(* Logix 5000 project; controller PLC2_Project_4_ServoApplication Emulate 5570 rev 20.11; software revision 20.00 *)
// A modular water treatment control system. Servo motor is connected to a cam/valve.

TASK MainTask (continuous, watchdog 500 ms) : MainProgram

MODULES
   Local : Emulate 5570 (ICP 1, rev 20.11)
      NicksIO : vendor 1 type 0 code 15 (ICP 2, rev 1.1, Output RPI 5 ms)
END_MODULES

PROGRAM MainProgram   (* main routine MainRoutine *)
VAR
   Button_CycleResetRequest : BOOL;
   Button_RequestCycle : BOOL;
   Cycle_Position : DINT := 4;   // Cycle Position/Mode 0 = Home 1 = Fill 2 = Drain 3 = Flush 4 = Travelling
   Cycle_Sequence : DINT := 3;   // Cycle Mode: SEQ 0 - FILL SEQ 1 - DRAIN SEQ 2 - FLUSH SEQ 3 - HOME
   DrainPosition_Delay : TIMER := (PRE := 20000);   // Drain position for 20 seconds
   FillPosition_Delay : TIMER := (PRE := 10000);   // Fill Position for 10 seconds
   FlushPosition_Delay : TIMER := (PRE := 10000);
   ONS_RequestCycle : BOOL;
   ONS_ResetRequest : BOOL;
   Servo_En : BOOL := 1;
   Switch_DrainPos : BOOL;
   Switch_FillPos : BOOL;
   Switch_FlushPos : BOOL;
   Switch_HomePos : BOOL;
END_VAR

ROUTINE Control   (* ladder *)
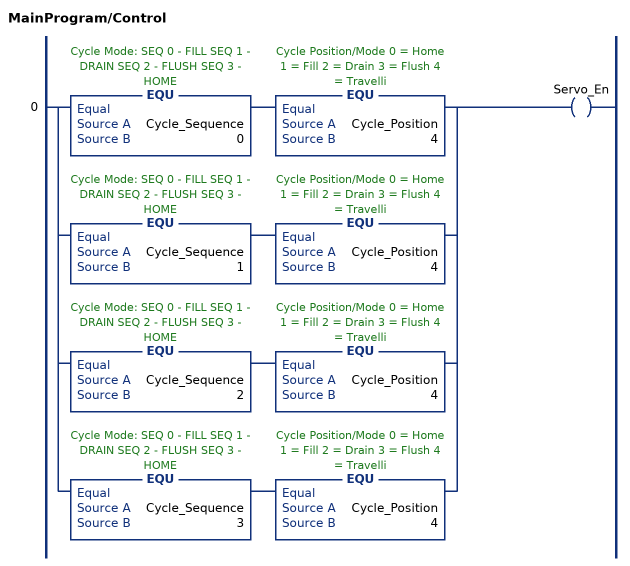
   0: [EQU(Cycle_Sequence,0) EQU(Cycle_Position,4) ,EQU(Cycle_Sequence,1) EQU(Cycle_Position,4) ,EQU(Cycle_Sequence,2) EQU(Cycle_Position,4) ,EQU(Cycle_Sequence,3) EQU(Cycle_Position,4) ]OTE(Servo_En);
END_ROUTINE

ROUTINE Cycle_Position   (* ladder *)
// What position is the valve in?
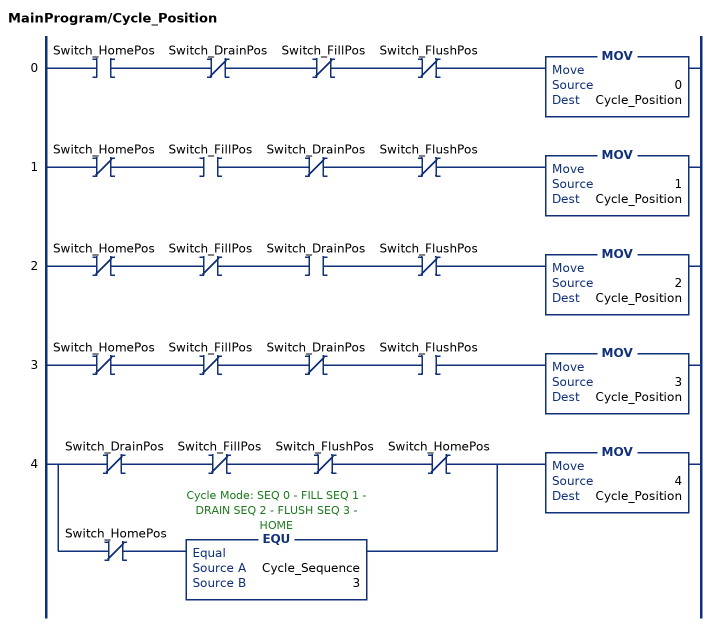
   0: XIC(Switch_HomePos)XIO(Switch_DrainPos)XIO(Switch_FillPos)XIO(Switch_FlushPos)MOV(0,Cycle_Position);
   1: XIO(Switch_HomePos)XIC(Switch_FillPos)XIO(Switch_DrainPos)XIO(Switch_FlushPos)MOV(1,Cycle_Position);
   2: XIO(Switch_HomePos)XIO(Switch_FillPos)XIC(Switch_DrainPos)XIO(Switch_FlushPos)MOV(2,Cycle_Position);
   3: XIO(Switch_HomePos)XIO(Switch_FillPos)XIO(Switch_DrainPos)XIC(Switch_FlushPos)MOV(3,Cycle_Position);
   4: [XIO(Switch_DrainPos) XIO(Switch_FillPos) XIO(Switch_FlushPos) XIO(Switch_HomePos) ,XIO(Switch_HomePos) EQU(Cycle_Sequence,3) ]MOV(4,Cycle_Position);
END_ROUTINE

ROUTINE Cycle_Sequence   (* ladder *)
// What stage in the cycle is the valve in?
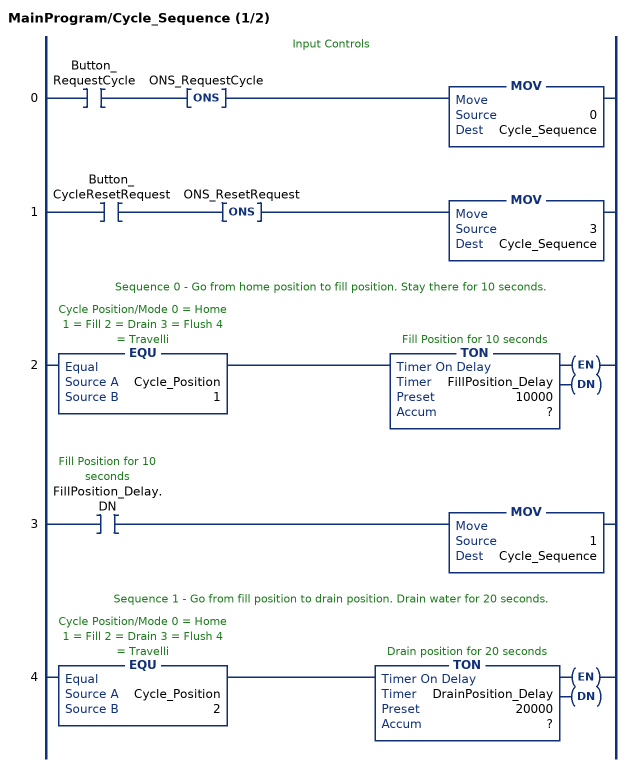
   // Input Controls
   0: XIC(Button_RequestCycle)ONS(ONS_RequestCycle)MOV(0,Cycle_Sequence);
   1: XIC(Button_CycleResetRequest)ONS(ONS_ResetRequest)MOV(3,Cycle_Sequence);
   // Sequence 0 - Go from home position to fill position. Stay there for 10 seconds.
   2: EQU(Cycle_Position,1)TON(FillPosition_Delay,?,?);
   3: XIC(FillPosition_Delay.DN)MOV(1,Cycle_Sequence);
   // Sequence 1 - Go from fill position to drain position. Drain water for 20 seconds.
   4: EQU(Cycle_Position,2)TON(DrainPosition_Delay,?,?);
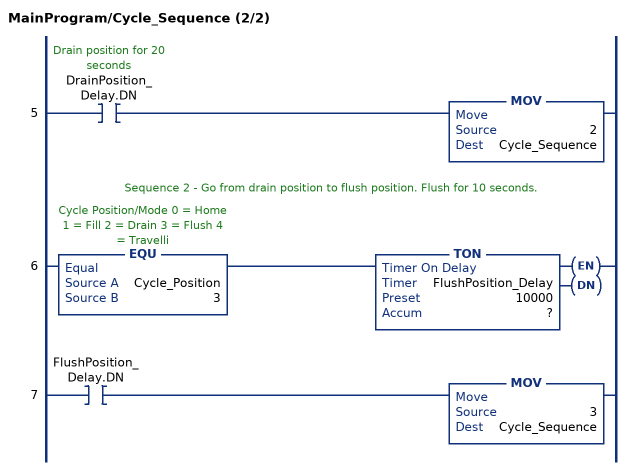
   5: XIC(DrainPosition_Delay.DN)MOV(2,Cycle_Sequence);
   // Sequence 2 - Go from drain position to flush position. Flush for 10 seconds.
   6: EQU(Cycle_Position,3)TON(FlushPosition_Delay,?,?);
   7: XIC(FlushPosition_Delay.DN)MOV(3,Cycle_Sequence);
END_ROUTINE

ROUTINE InputOutput   (* ladder *)
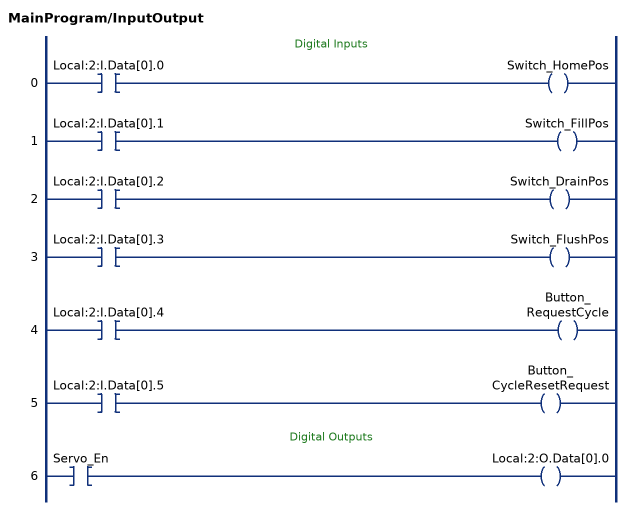
   // Digital Inputs
   0: XIC(Local:2:I.Data[0].0)OTE(Switch_HomePos);
   1: XIC(Local:2:I.Data[0].1)OTE(Switch_FillPos);
   2: XIC(Local:2:I.Data[0].2)OTE(Switch_DrainPos);
   3: XIC(Local:2:I.Data[0].3)OTE(Switch_FlushPos);
   4: XIC(Local:2:I.Data[0].4)OTE(Button_RequestCycle);
   5: XIC(Local:2:I.Data[0].5)OTE(Button_CycleResetRequest);
   // Digital Outputs
   6: XIC(Servo_En)OTE(Local:2:O.Data[0].0);
END_ROUTINE

ROUTINE MainRoutine   (* ladder *)
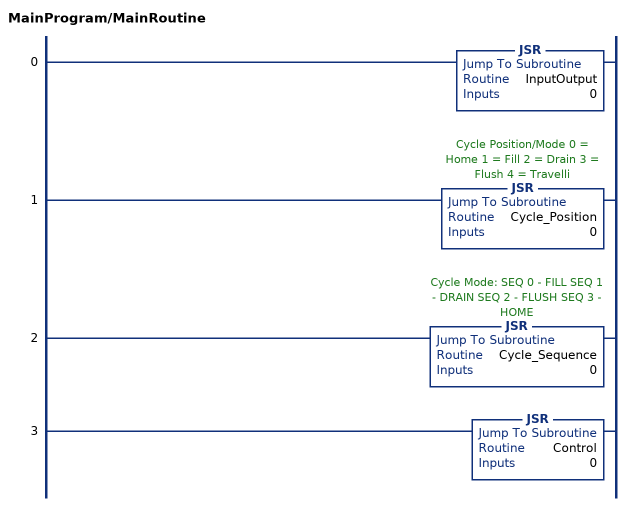
   0: JSR(InputOutput,0);
   1: JSR(Cycle_Position,0);
   2: JSR(Cycle_Sequence,0);
   3: JSR(Control,0);
END_ROUTINE
END_PROGRAM
